// TIA Portal V20 export
VAR_GLOBAL   // PLC tag table "Default tag table"
   Tag_1 AT %M2.1 : Bool;
   toto AT %M2.2 : Bool;
   Tag_2 AT %M0.0 : Bool;
END_VAR
